# EPICS substitutions: aldn1000Sup/unit_setter.substitutions
file $(UTILITIES)/db/unit_setter.template {
  pattern
    {P,    FROM, TO}

    {"\$(P)", "VOLUME:UNITS", "VOLUME"}
    {"\$(P)", "VOLUME:UNITS", "VOLUME:SP"}
    {"\$(P)", "VOLUME:UNITS", "VOLUME:INF"}
    {"\$(P)", "VOLUME:UNITS", "VOLUME:WDR"}

    {"\$(P)", "RATE:UNITS", "RATE"}
    {"\$(P)", "RATE:UNITS", "RATE:SP"}
}
